FUNCTION_BLOCK CONTROL_CHART
  {SET_ATTRIBUTE(OpcUa, SERVICE)}
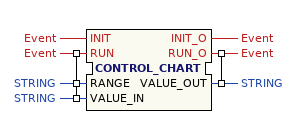
  EVENT_INPUT
    INIT;
    RUN WITH RANGE, VALUE_IN;
  END_EVENT
  EVENT_OUTPUT
    INIT_O;
    RUN_O WITH VALUE_OUT;
  END_EVENT
  VAR_INPUT
    RANGE : STRING; {SET_ATTRIBUTE(OpcUa, Constant)}
    VALUE_IN : STRING; {SET_ATTRIBUTE(OpcUa, Variable)}
  END_VAR
  VAR_OUTPUT
    VALUE_OUT : STRING; {SET_ATTRIBUTE(OpcUa, Variable)}
  END_VAR
END_FUNCTION_BLOCK
